FUNCTION_BLOCK TO_CNV_MODEL (* Composite Function Block Type *)
  (* Standard: 61499-2 *)
  (* Version 0.2, 2003-12-05, JHC, Rockwell Automation, Renamed from NEWCOMPFB. *)
  (* Version 0.1, 2002-01-08, JHC, Rockwell Automation, Added DLY FB as example. *)
  (* Version 0.0, 2000-05-27, JHC, Rockwell Automation *)
  (* Compiler header: package fb.rt.template; *)
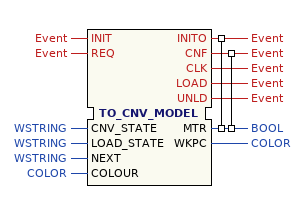
  EVENT_INPUT
    INIT; (* Initialization Request *)
    REQ; (* Normal Execution Request *)
  END_EVENT
  EVENT_OUTPUT
    INITO WITH MTR; (* Initialization Confirm *)
    CNF WITH MTR; (* Execution Confirmation *)
    CLK;
    LOAD;
    UNLD;
  END_EVENT
  VAR_INPUT
    CNV_STATE : WSTRING;
    LOAD_STATE : WSTRING;
    NEXT : WSTRING;
    COLOUR : COLOR;
  END_VAR
  VAR_OUTPUT
    MTR : BOOL; (* Output event qualifier *)
    WKPC : COLOR;
  END_VAR
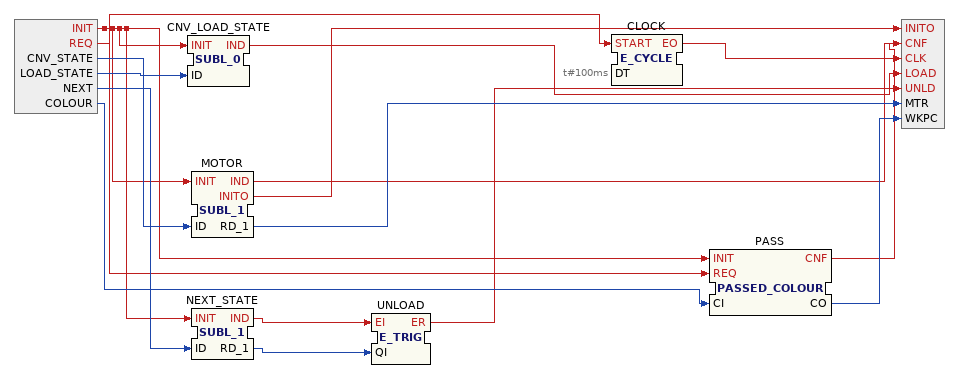
  FBS
    MOTOR : SUBL_1;
    CNV_LOAD_STATE : SUBL_0;
    NEXT_STATE : SUBL_1;
    UNLOAD : E_TRIG;
    CLOCK : E_CYCLE(DT := t#100ms);
    PASS : PASSED_COLOUR;
  END_FBS
  EVENT_CONNECTIONS
    INIT TO MOTOR.INIT;
    INIT TO CNV_LOAD_STATE.INIT;
    INIT TO NEXT_STATE.INIT;
    NEXT_STATE.IND TO UNLOAD.EI;
    CLOCK.EO TO CLK;
    REQ TO CLOCK.START;
    CNV_LOAD_STATE.IND TO LOAD;
    UNLOAD.ER TO UNLD;
    MOTOR.IND TO CNF;
    MOTOR.INITO TO INITO;
    INIT TO PASS.INIT;
    REQ TO PASS.REQ;
    PASS.CNF TO CNF;
  END_CONNECTIONS
  DATA_CONNECTIONS
    NEXT_STATE.RD_1 TO UNLOAD.QI;
    LOAD_STATE TO CNV_LOAD_STATE.ID;
    CNV_STATE TO MOTOR.ID;
    NEXT TO NEXT_STATE.ID;
    MOTOR.RD_1 TO MTR;
    COLOUR TO PASS.CI;
    PASS.CO TO WKPC;
  END_CONNECTIONS
END_FUNCTION_BLOCK
